TEXTLIST visuTextLinks_1
  A = 'GVL.axes[1].Axis.NcToPlc.ActPos'
   = ''
END_TEXTLIST

(* stored: Version 1.1.0.1, ProductVersion 3.1.4024.0
   TextList visuTextLinks_1: Id {c78aee74-a2f6-4c8e-a8d0-d0d31eec8cd3} *)
